{attribute addProperty BoxType "AX8620-1000-0027"}
{attribute addProperty Id "PSM_PSM_StatuswordAT %I*PSM_PSM_Statusword_C154CB391620WcStateAT %I*WcState_F855686C1620InfoDataAT %I*InfoData_0BDED7BF144180"}
{attribute addProperty CRC "4282750922"}
{attribute addProperty SizeInBites "176"}
{attribute addProperty SizeInBytes "22"}
TYPE AX8620_A1A6213B :
STRUCT
	{attribute addProperty Name "PSM_PSM_Statusword"}
	PSM_PSM_Statusword : PSM_PSM_Statusword_C154CB39;
	{attribute addProperty Name "WcState"}
	WcState : WcState_F855686C;
	{attribute addProperty Name "InfoData"}
	InfoData : InfoData_0BDED7BF;
END_STRUCT
END_TYPE

(* stored: Version 1.2.0.0, ProductVersion 3.1.4024.9
   DUT AX8620_A1A6213B: Id {df94fa24-3076-424e-a21b-7716ca3b6808} *)
